// TwinCAT 3 PLC project TestIOC
// ProgramVersion: 3.1.4026.17
// libraries:
//   LCLS General, * (SLAC)
//   LCLS Vacuum, * (SLAC - LCLS)
//   lcls-twincat-common-components, * (SLAC)
//   lcls-twincat-math, * (SLAC - LCLS)
//   lcls-twincat-motion, * (SLAC)
//   lcls-twincat-optics, * (SLAC)
//   lcls-twincat-physics, * (SLAC)
//   LCLS_MotionAbstraction, * (SLAC)
//   LCLS_Tc_DevAbs, * (SLAC - LCLS)
//   PMPS, * (SLAC - LCLS)
//   Tc2_MC2, * (Beckhoff Automation GmbH)
//   Tc2_Standard, * (Beckhoff Automation GmbH)
//   Tc2_System, * (Beckhoff Automation GmbH)
//   Tc3_Module, * (Beckhoff Automation GmbH)
//   TcUnit, * (www.tcunit.org)
// project tree:
//   DUTs/ ENUM_Test.TcDUT (not stored), ST_NestedTypes01.TcDUT, ST_NestedTypes02.TcDUT, ST_NestedTypes03.TcDUT, ST_NestedTypes04.TcDUT, ST_NestedTypes05.TcDUT, ST_PytmcTypes.TcDUT (not stored)
//   GVLs/ GVL.TcGVL
//   / PlcTask.TcTTO
//   POUs/ Main.TcPOU (not stored), F_UpdateArray.TcPOU (not stored)
// real-time tasks:
//   TASK PlcTask: cycle T#10ms, priority 20, ADS port 350
// motion (NC):
//   TASK NC-Task 1 SAF: cycle T#2ms, priority 4, ADS port 501
//   TASK NC-Task 1 SVB: cycle T#10ms, priority 8, ADS port 511
//   AXIS Axis 1 (id 1)
//     OtherSettings: AllowMotionCmdToSlave=true
//     encoder EncType=1
//     drive DrvType=5
//       Analog: TorqueSetpointScale=10, ScaleFactorActTorque=0.1
//       TimeComp: TaskDelayCycles=1
//     controller CtrType=1
//       CtrPara: PriorControlFactor=1
//         Observer: BandWidth=20
//   AXIS Axis 2 (id 2)
//     OtherSettings: AllowMotionCmdToSlave=true
//     encoder EncType=1
//     drive DrvType=5
//       Analog: TorqueSetpointScale=10, ScaleFactorActTorque=0.1
//       TimeComp: TaskDelayCycles=1
//     controller CtrType=1
//       CtrPara: PriorControlFactor=1
//         Observer: BandWidth=20
//   AXIS Axis 3 (id 3)
//     OtherSettings: AllowMotionCmdToSlave=true
//     encoder EncType=1
//     drive DrvType=5
//       Analog: TorqueSetpointScale=10, ScaleFactorActTorque=0.1
//       TimeComp: TaskDelayCycles=1
//     controller CtrType=1
//       CtrPara: PriorControlFactor=1
//         Observer: BandWidth=20
//   AXIS Axis 4 (id 4)
//     OtherSettings: AllowMotionCmdToSlave=true
//     encoder EncType=1
//     drive DrvType=5
//       Analog: TorqueSetpointScale=10, ScaleFactorActTorque=0.1
//       TimeComp: TaskDelayCycles=1
//     controller CtrType=1
//       CtrPara: PriorControlFactor=1
//         Observer: BandWidth=20
//   AXIS Axis 5 (id 5)
//     OtherSettings: AllowMotionCmdToSlave=true
//     encoder EncType=1
//     drive DrvType=5
//       Analog: TorqueSetpointScale=10, ScaleFactorActTorque=0.1
//       TimeComp: TaskDelayCycles=1
//     controller CtrType=1
//       CtrPara: PriorControlFactor=1
//         Observer: BandWidth=20
//   AXIS Axis 6 (id 6)
//     OtherSettings: AllowMotionCmdToSlave=true
//     encoder EncType=1
//     drive DrvType=5
//       Analog: TorqueSetpointScale=10, ScaleFactorActTorque=0.1
//       TimeComp: TaskDelayCycles=1
//     controller CtrType=1
//       CtrPara: PriorControlFactor=1
//         Observer: BandWidth=20
//   AXIS Axis 7 (id 7)
//     OtherSettings: AllowMotionCmdToSlave=true
//     encoder EncType=1
//     drive DrvType=5
//       Analog: TorqueSetpointScale=10, ScaleFactorActTorque=0.1
//       TimeComp: TaskDelayCycles=1
//     controller CtrType=1
//       CtrPara: PriorControlFactor=1
//         Observer: BandWidth=20
//   AXIS Axis 8 (id 8)
//     OtherSettings: AllowMotionCmdToSlave=true
//     encoder EncType=1
//     drive DrvType=5
//       Analog: TorqueSetpointScale=10, ScaleFactorActTorque=0.1
//       TimeComp: TaskDelayCycles=1
//     controller CtrType=1
//       CtrPara: PriorControlFactor=1
//         Observer: BandWidth=20
//   AXIS Axis 9 (id 9)
//     OtherSettings: AllowMotionCmdToSlave=true
//     encoder EncType=1
//     drive DrvType=5
//       Analog: TorqueSetpointScale=10, ScaleFactorActTorque=0.1
//       TimeComp: TaskDelayCycles=1
//     controller CtrType=1
//       CtrPara: PriorControlFactor=1
//         Observer: BandWidth=20
//   AXIS Axis 10 (id 10)
//     OtherSettings: AllowMotionCmdToSlave=true
//     encoder EncType=1
//     drive DrvType=5
//       Analog: TorqueSetpointScale=10, ScaleFactorActTorque=0.1
//       TimeComp: TaskDelayCycles=1
//     controller CtrType=1
//       CtrPara: PriorControlFactor=1
//         Observer: BandWidth=20
//   AXIS Axis 11 (id 11)
//     OtherSettings: AllowMotionCmdToSlave=true
//     encoder EncType=1
//     drive DrvType=5
//       Analog: TorqueSetpointScale=10, ScaleFactorActTorque=0.1
//       TimeComp: TaskDelayCycles=1
//     controller CtrType=1
//       CtrPara: PriorControlFactor=1
//         Observer: BandWidth=20
//   AXIS Axis 12 (id 12)
//     OtherSettings: AllowMotionCmdToSlave=true
//     encoder EncType=1
//     drive DrvType=5
//       Analog: TorqueSetpointScale=10, ScaleFactorActTorque=0.1
//       TimeComp: TaskDelayCycles=1
//     controller CtrType=1
//       CtrPara: PriorControlFactor=1
//         Observer: BandWidth=20
//   AXIS Axis 13 (id 13)
//     OtherSettings: AllowMotionCmdToSlave=true
//     encoder EncType=1
//     drive DrvType=5
//       Analog: TorqueSetpointScale=10, ScaleFactorActTorque=0.1
//       TimeComp: TaskDelayCycles=1
//     controller CtrType=1
//       CtrPara: PriorControlFactor=1
//         Observer: BandWidth=20
//   AXIS Axis 14 (id 14)
//     OtherSettings: AllowMotionCmdToSlave=true
//     encoder EncType=1
//     drive DrvType=5
//       Analog: TorqueSetpointScale=10, ScaleFactorActTorque=0.1
//       TimeComp: TaskDelayCycles=1
//     controller CtrType=1
//       CtrPara: PriorControlFactor=1
//         Observer: BandWidth=20
//   AXIS Axis 15 (id 15)
//     OtherSettings: AllowMotionCmdToSlave=true
//     encoder EncType=1
//     drive DrvType=5
//       Analog: TorqueSetpointScale=10, ScaleFactorActTorque=0.1
//       TimeComp: TaskDelayCycles=1
//     controller CtrType=1
//       CtrPara: PriorControlFactor=1
//         Observer: BandWidth=20
//   AXIS Axis 16 (id 16)
//     OtherSettings: AllowMotionCmdToSlave=true
//     encoder EncType=1
//     drive DrvType=5
//       Analog: TorqueSetpointScale=10, ScaleFactorActTorque=0.1
//       TimeComp: TaskDelayCycles=1
//     controller CtrType=1
//       CtrPara: PriorControlFactor=1
//         Observer: BandWidth=20
//   AXIS Axis 17 (id 17)
//     OtherSettings: AllowMotionCmdToSlave=true
//     encoder EncType=1
//     drive DrvType=5
//       Analog: TorqueSetpointScale=10, ScaleFactorActTorque=0.1
//       TimeComp: TaskDelayCycles=1
//     controller CtrType=1
//       CtrPara: PriorControlFactor=1
//         Observer: BandWidth=20
//   AXIS Axis 18 (id 18)
//     OtherSettings: AllowMotionCmdToSlave=true
//     encoder EncType=1
//     drive DrvType=5
//       Analog: TorqueSetpointScale=10, ScaleFactorActTorque=0.1
//       TimeComp: TaskDelayCycles=1
//     controller CtrType=1
//       CtrPara: PriorControlFactor=1
//         Observer: BandWidth=20
//   AXIS Axis 19 (id 19)
//     OtherSettings: AllowMotionCmdToSlave=true
//     encoder EncType=1
//     drive DrvType=5
//       Analog: TorqueSetpointScale=10, ScaleFactorActTorque=0.1
//       TimeComp: TaskDelayCycles=1
//     controller CtrType=1
//       CtrPara: PriorControlFactor=1
//         Observer: BandWidth=20
//   AXIS Axis 20 (id 20)
//     OtherSettings: AllowMotionCmdToSlave=true
//     encoder EncType=1
//     drive DrvType=5
//       Analog: TorqueSetpointScale=10, ScaleFactorActTorque=0.1
//       TimeComp: TaskDelayCycles=1
//     controller CtrType=1
//       CtrPara: PriorControlFactor=1
//         Observer: BandWidth=20
//   AXIS Axis 21 (id 21)
//     OtherSettings: AllowMotionCmdToSlave=true
//     encoder EncType=1
//     drive DrvType=5
//       Analog: TorqueSetpointScale=10, ScaleFactorActTorque=0.1
//       TimeComp: TaskDelayCycles=1
//     controller CtrType=1
//       CtrPara: PriorControlFactor=1
//         Observer: BandWidth=20
//   AXIS Axis 22 (id 22)
//     OtherSettings: AllowMotionCmdToSlave=true
//     encoder EncType=1
//     drive DrvType=5
//       Analog: TorqueSetpointScale=10, ScaleFactorActTorque=0.1
//       TimeComp: TaskDelayCycles=1
//     controller CtrType=1
//       CtrPara: PriorControlFactor=1
//         Observer: BandWidth=20
//   AXIS Axis 23 (id 23)
//     OtherSettings: AllowMotionCmdToSlave=true
//     encoder EncType=1
//     drive DrvType=5
//       Analog: TorqueSetpointScale=10, ScaleFactorActTorque=0.1
//       TimeComp: TaskDelayCycles=1
//     controller CtrType=1
//       CtrPara: PriorControlFactor=1
//         Observer: BandWidth=20
//   AXIS Axis 24 (id 24)
//     OtherSettings: AllowMotionCmdToSlave=true
//     encoder EncType=1
//     drive DrvType=5
//       Analog: TorqueSetpointScale=10, ScaleFactorActTorque=0.1
//       TimeComp: TaskDelayCycles=1
//     controller CtrType=1
//       CtrPara: PriorControlFactor=1
//         Observer: BandWidth=20
//   AXIS Axis 25 (id 25)
//     OtherSettings: AllowMotionCmdToSlave=true
//     encoder EncType=1
//     drive DrvType=5
//       Analog: TorqueSetpointScale=10, ScaleFactorActTorque=0.1
//       TimeComp: TaskDelayCycles=1
//     controller CtrType=1
//       CtrPara: PriorControlFactor=1
//         Observer: BandWidth=20
//   AXIS Axis 26 (id 26)
//     OtherSettings: AllowMotionCmdToSlave=true
//     encoder EncType=1
//     drive DrvType=5
//       Analog: TorqueSetpointScale=10, ScaleFactorActTorque=0.1
//       TimeComp: TaskDelayCycles=1
//     controller CtrType=1
//       CtrPara: PriorControlFactor=1
//         Observer: BandWidth=20
//   AXIS Axis 27 (id 27)
//     OtherSettings: AllowMotionCmdToSlave=true
//     encoder EncType=1
//     drive DrvType=5
//       Analog: TorqueSetpointScale=10, ScaleFactorActTorque=0.1
//       TimeComp: TaskDelayCycles=1
//     controller CtrType=1
//       CtrPara: PriorControlFactor=1
//         Observer: BandWidth=20
//   AXIS Axis 28 (id 28)
//     OtherSettings: AllowMotionCmdToSlave=true
//     encoder EncType=1
//     drive DrvType=5
//       Analog: TorqueSetpointScale=10, ScaleFactorActTorque=0.1
//       TimeComp: TaskDelayCycles=1
//     controller CtrType=1
//       CtrPara: PriorControlFactor=1
//         Observer: BandWidth=20
//   AXIS Axis 29 (id 29)
//     OtherSettings: AllowMotionCmdToSlave=true
//     encoder EncType=1
//     drive DrvType=5
//       Analog: TorqueSetpointScale=10, ScaleFactorActTorque=0.1
//       TimeComp: TaskDelayCycles=1
//     controller CtrType=1
//       CtrPara: PriorControlFactor=1
//         Observer: BandWidth=20
//   AXIS Axis 30 (id 30)
//     OtherSettings: AllowMotionCmdToSlave=true
//     encoder EncType=1
//     drive DrvType=5
//       Analog: TorqueSetpointScale=10, ScaleFactorActTorque=0.1
//       TimeComp: TaskDelayCycles=1
//     controller CtrType=1
//       CtrPara: PriorControlFactor=1
//         Observer: BandWidth=20
//   AXIS Axis 31 (id 31)
//     OtherSettings: AllowMotionCmdToSlave=true
//     encoder EncType=1
//     drive DrvType=5
//       Analog: TorqueSetpointScale=10, ScaleFactorActTorque=0.1
//       TimeComp: TaskDelayCycles=1
//     controller CtrType=1
//       CtrPara: PriorControlFactor=1
//         Observer: BandWidth=20
//   AXIS Axis 32 (id 32)
//     OtherSettings: AllowMotionCmdToSlave=true
//     encoder EncType=1
//     drive DrvType=5
//       Analog: TorqueSetpointScale=10, ScaleFactorActTorque=0.1
//       TimeComp: TaskDelayCycles=1
//     controller CtrType=1
//       CtrPara: PriorControlFactor=1
//         Observer: BandWidth=20
//   AXIS Axis 33 (id 33)
//     OtherSettings: AllowMotionCmdToSlave=true
//     encoder EncType=1
//     drive DrvType=5
//       Analog: TorqueSetpointScale=10, ScaleFactorActTorque=0.1
//       TimeComp: TaskDelayCycles=1
//     controller CtrType=1
//       CtrPara: PriorControlFactor=1
//         Observer: BandWidth=20
//   AXIS Axis 34 (id 34)
//     OtherSettings: AllowMotionCmdToSlave=true
//     encoder EncType=1
//     drive DrvType=5
//       Analog: TorqueSetpointScale=10, ScaleFactorActTorque=0.1
//       TimeComp: TaskDelayCycles=1
//     controller CtrType=1
//       CtrPara: PriorControlFactor=1
//         Observer: BandWidth=20
//   AXIS Axis 35 (id 35)
//     OtherSettings: AllowMotionCmdToSlave=true
//     encoder EncType=1
//     drive DrvType=5
//       Analog: TorqueSetpointScale=10, ScaleFactorActTorque=0.1
//       TimeComp: TaskDelayCycles=1
//     controller CtrType=1
//       CtrPara: PriorControlFactor=1
//         Observer: BandWidth=20
//   AXIS Axis 36 (id 36)
//     OtherSettings: AllowMotionCmdToSlave=true
//     encoder EncType=1
//     drive DrvType=5
//       Analog: TorqueSetpointScale=10, ScaleFactorActTorque=0.1
//       TimeComp: TaskDelayCycles=1
//     controller CtrType=1
//       CtrPara: PriorControlFactor=1
//         Observer: BandWidth=20
//   AXIS Axis 37 (id 37)
//     OtherSettings: AllowMotionCmdToSlave=true
//     encoder EncType=1
//     drive DrvType=5
//       Analog: TorqueSetpointScale=10, ScaleFactorActTorque=0.1
//       TimeComp: TaskDelayCycles=1
//     controller CtrType=1
//       CtrPara: PriorControlFactor=1
//         Observer: BandWidth=20
//   AXIS Axis 38 (id 38)
//     OtherSettings: AllowMotionCmdToSlave=true
//     encoder EncType=1
//     drive DrvType=5
//       Analog: TorqueSetpointScale=10, ScaleFactorActTorque=0.1
//       TimeComp: TaskDelayCycles=1
//     controller CtrType=1
//       CtrPara: PriorControlFactor=1
//         Observer: BandWidth=20
//   AXIS Axis 39 (id 39)
//     OtherSettings: AllowMotionCmdToSlave=true
//     encoder EncType=1
//     drive DrvType=5
//       Analog: TorqueSetpointScale=10, ScaleFactorActTorque=0.1
//       TimeComp: TaskDelayCycles=1
//     controller CtrType=1
//       CtrPara: PriorControlFactor=1
//         Observer: BandWidth=20
//   AXIS Axis 40 (id 40)
//     OtherSettings: AllowMotionCmdToSlave=true
//     encoder EncType=1
//     drive DrvType=5
//       Analog: TorqueSetpointScale=10, ScaleFactorActTorque=0.1
//       TimeComp: TaskDelayCycles=1
//     controller CtrType=1
//       CtrPara: PriorControlFactor=1
//         Observer: BandWidth=20
//   AXIS Axis 41 (id 41)
//     OtherSettings: AllowMotionCmdToSlave=true
//     encoder EncType=1
//     drive DrvType=5
//       Analog: TorqueSetpointScale=10, ScaleFactorActTorque=0.1
//       TimeComp: TaskDelayCycles=1
//     controller CtrType=1
//       CtrPara: PriorControlFactor=1
//         Observer: BandWidth=20
//   AXIS Axis 42 (id 42)
//     OtherSettings: AllowMotionCmdToSlave=true
//     encoder EncType=1
//     drive DrvType=5
//       Analog: TorqueSetpointScale=10, ScaleFactorActTorque=0.1
//       TimeComp: TaskDelayCycles=1
//     controller CtrType=1
//       CtrPara: PriorControlFactor=1
//         Observer: BandWidth=20
//   AXIS Axis 43 (id 43)
//     OtherSettings: AllowMotionCmdToSlave=true
//     encoder EncType=1
//     drive DrvType=5
//       Analog: TorqueSetpointScale=10, ScaleFactorActTorque=0.1
//       TimeComp: TaskDelayCycles=1
//     controller CtrType=1
//       CtrPara: PriorControlFactor=1
//         Observer: BandWidth=20
//   AXIS Axis 44 (id 44)
//     OtherSettings: AllowMotionCmdToSlave=true
//     encoder EncType=1
//     drive DrvType=5
//       Analog: TorqueSetpointScale=10, ScaleFactorActTorque=0.1
//       TimeComp: TaskDelayCycles=1
//     controller CtrType=1
//       CtrPara: PriorControlFactor=1
//         Observer: BandWidth=20
//   AXIS Axis 45 (id 45)
//     OtherSettings: AllowMotionCmdToSlave=true
//     encoder EncType=1
//     drive DrvType=5
//       Analog: TorqueSetpointScale=10, ScaleFactorActTorque=0.1
//       TimeComp: TaskDelayCycles=1
//     controller CtrType=1
//       CtrPara: PriorControlFactor=1
//         Observer: BandWidth=20
//   AXIS Axis 46 (id 46)
//     OtherSettings: AllowMotionCmdToSlave=true
//     encoder EncType=1
//     drive DrvType=5
//       Analog: TorqueSetpointScale=10, ScaleFactorActTorque=0.1
//       TimeComp: TaskDelayCycles=1
//     controller CtrType=1
//       CtrPara: PriorControlFactor=1
//         Observer: BandWidth=20
//   AXIS Axis 47 (id 47)
//     OtherSettings: AllowMotionCmdToSlave=true
//     encoder EncType=1
//     drive DrvType=5
//       Analog: TorqueSetpointScale=10, ScaleFactorActTorque=0.1
//       TimeComp: TaskDelayCycles=1
//     controller CtrType=1
//       CtrPara: PriorControlFactor=1
//         Observer: BandWidth=20
//   AXIS Axis 48 (id 48)
//     OtherSettings: AllowMotionCmdToSlave=true
//     encoder EncType=1
//     drive DrvType=5
//       Analog: TorqueSetpointScale=10, ScaleFactorActTorque=0.1
//       TimeComp: TaskDelayCycles=1
//     controller CtrType=1
//       CtrPara: PriorControlFactor=1
//         Observer: BandWidth=20
//   AXIS Axis 49 (id 49)
//     OtherSettings: AllowMotionCmdToSlave=true
//     encoder EncType=1
//     drive DrvType=5
//       Analog: TorqueSetpointScale=10, ScaleFactorActTorque=0.1
//       TimeComp: TaskDelayCycles=1
//     controller CtrType=1
//       CtrPara: PriorControlFactor=1
//         Observer: BandWidth=20
//   AXIS Axis 50 (id 50)
//     OtherSettings: AllowMotionCmdToSlave=true
//     encoder EncType=1
//     drive DrvType=5
//       Analog: TorqueSetpointScale=10, ScaleFactorActTorque=0.1
//       TimeComp: TaskDelayCycles=1
//     controller CtrType=1
//       CtrPara: PriorControlFactor=1
//         Observer: BandWidth=20
//   AXIS Axis 51 (id 51)
//     OtherSettings: AllowMotionCmdToSlave=true
//     encoder EncType=1
//     drive DrvType=5
//       Analog: TorqueSetpointScale=10, ScaleFactorActTorque=0.1
//       TimeComp: TaskDelayCycles=1
//     controller CtrType=1
//       CtrPara: PriorControlFactor=1
//         Observer: BandWidth=20
//   AXIS Axis 52 (id 52)
//     OtherSettings: AllowMotionCmdToSlave=true
//     encoder EncType=1
//     drive DrvType=5
//       Analog: TorqueSetpointScale=10, ScaleFactorActTorque=0.1
//       TimeComp: TaskDelayCycles=1
//     controller CtrType=1
//       CtrPara: PriorControlFactor=1
//         Observer: BandWidth=20
// variable links:
//   (this object) <-> NC-Task 1 SAF/Axes/Axis 1
//     PlcTask Inputs/Main.M1.Axis.NcToPlc <-> Outputs/ToPlc
//     PlcTask Outputs/Main.M1.Axis.PlcToNc <-> Inputs/FromPlc
//   (this object) <-> NC-Task 1 SAF/Axes/Axis 10
//     PlcTask Inputs/Main.aAxisRef[8].NcToPlc <-> Outputs/ToPlc
//     PlcTask Outputs/Main.aAxisRef[8].PlcToNc <-> Inputs/FromPlc
//   (this object) <-> NC-Task 1 SAF/Axes/Axis 11
//     PlcTask Inputs/Main.aAxisRef[9].NcToPlc <-> Outputs/ToPlc
//     PlcTask Outputs/Main.aAxisRef[9].PlcToNc <-> Inputs/FromPlc
//   (this object) <-> NC-Task 1 SAF/Axes/Axis 12
//     PlcTask Inputs/Main.aAxisRef[10].NcToPlc <-> Outputs/ToPlc
//     PlcTask Outputs/Main.aAxisRef[10].PlcToNc <-> Inputs/FromPlc
//   (this object) <-> NC-Task 1 SAF/Axes/Axis 13
//     PlcTask Inputs/Main.aAxisRef[11].NcToPlc <-> Outputs/ToPlc
//     PlcTask Outputs/Main.aAxisRef[11].PlcToNc <-> Inputs/FromPlc
//   (this object) <-> NC-Task 1 SAF/Axes/Axis 14
//     PlcTask Inputs/Main.aAxisRef[12].NcToPlc <-> Outputs/ToPlc
//     PlcTask Outputs/Main.aAxisRef[12].PlcToNc <-> Inputs/FromPlc
//   (this object) <-> NC-Task 1 SAF/Axes/Axis 15
//     PlcTask Inputs/Main.aAxisRef[13].NcToPlc <-> Outputs/ToPlc
//     PlcTask Outputs/Main.aAxisRef[13].PlcToNc <-> Inputs/FromPlc
//   (this object) <-> NC-Task 1 SAF/Axes/Axis 16
//     PlcTask Inputs/Main.aAxisRef[14].NcToPlc <-> Outputs/ToPlc
//     PlcTask Outputs/Main.aAxisRef[14].PlcToNc <-> Inputs/FromPlc
//   (this object) <-> NC-Task 1 SAF/Axes/Axis 17
//     PlcTask Inputs/Main.aAxisRef[15].NcToPlc <-> Outputs/ToPlc
//     PlcTask Outputs/Main.aAxisRef[15].PlcToNc <-> Inputs/FromPlc
//   (this object) <-> NC-Task 1 SAF/Axes/Axis 18
//     PlcTask Inputs/Main.aAxisRef[16].NcToPlc <-> Outputs/ToPlc
//     PlcTask Outputs/Main.aAxisRef[16].PlcToNc <-> Inputs/FromPlc
//   (this object) <-> NC-Task 1 SAF/Axes/Axis 19
//     PlcTask Inputs/Main.aAxisRef[17].NcToPlc <-> Outputs/ToPlc
//     PlcTask Outputs/Main.aAxisRef[17].PlcToNc <-> Inputs/FromPlc
//   (this object) <-> NC-Task 1 SAF/Axes/Axis 2
//     PlcTask Inputs/Main.M2.Axis.NcToPlc <-> Outputs/ToPlc
//     PlcTask Outputs/Main.M2.Axis.PlcToNc <-> Inputs/FromPlc
//   (this object) <-> NC-Task 1 SAF/Axes/Axis 20
//     PlcTask Inputs/Main.aAxisRef[18].NcToPlc <-> Outputs/ToPlc
//     PlcTask Outputs/Main.aAxisRef[18].PlcToNc <-> Inputs/FromPlc
//   (this object) <-> NC-Task 1 SAF/Axes/Axis 21
//     PlcTask Inputs/Main.aAxisRef[19].NcToPlc <-> Outputs/ToPlc
//     PlcTask Outputs/Main.aAxisRef[19].PlcToNc <-> Inputs/FromPlc
//   (this object) <-> NC-Task 1 SAF/Axes/Axis 22
//     PlcTask Inputs/Main.aAxisRef[20].NcToPlc <-> Outputs/ToPlc
//     PlcTask Outputs/Main.aAxisRef[20].PlcToNc <-> Inputs/FromPlc
//   (this object) <-> NC-Task 1 SAF/Axes/Axis 23
//     PlcTask Inputs/Main.aAxisRef[21].NcToPlc <-> Outputs/ToPlc
//     PlcTask Outputs/Main.aAxisRef[21].PlcToNc <-> Inputs/FromPlc
//   (this object) <-> NC-Task 1 SAF/Axes/Axis 24
//     PlcTask Inputs/Main.aAxisRef[22].NcToPlc <-> Outputs/ToPlc
//     PlcTask Outputs/Main.aAxisRef[22].PlcToNc <-> Inputs/FromPlc
//   (this object) <-> NC-Task 1 SAF/Axes/Axis 25
//     PlcTask Inputs/Main.aAxisRef[23].NcToPlc <-> Outputs/ToPlc
//     PlcTask Outputs/Main.aAxisRef[23].PlcToNc <-> Inputs/FromPlc
//   (this object) <-> NC-Task 1 SAF/Axes/Axis 26
//     PlcTask Inputs/Main.aAxisRef[24].NcToPlc <-> Outputs/ToPlc
//     PlcTask Outputs/Main.aAxisRef[24].PlcToNc <-> Inputs/FromPlc
//   (this object) <-> NC-Task 1 SAF/Axes/Axis 27
//     PlcTask Inputs/Main.aAxisRef[25].NcToPlc <-> Outputs/ToPlc
//     PlcTask Outputs/Main.aAxisRef[25].PlcToNc <-> Inputs/FromPlc
//   (this object) <-> NC-Task 1 SAF/Axes/Axis 28
//     PlcTask Inputs/Main.aAxisRef[26].NcToPlc <-> Outputs/ToPlc
//     PlcTask Outputs/Main.aAxisRef[26].PlcToNc <-> Inputs/FromPlc
//   (this object) <-> NC-Task 1 SAF/Axes/Axis 29
//     PlcTask Inputs/Main.aAxisRef[27].NcToPlc <-> Outputs/ToPlc
//     PlcTask Outputs/Main.aAxisRef[27].PlcToNc <-> Inputs/FromPlc
//   (this object) <-> NC-Task 1 SAF/Axes/Axis 3
//     PlcTask Inputs/Main.aAxisRef[1].NcToPlc <-> Outputs/ToPlc
//     PlcTask Outputs/Main.aAxisRef[1].PlcToNc <-> Inputs/FromPlc
//   (this object) <-> NC-Task 1 SAF/Axes/Axis 30
//     PlcTask Inputs/Main.aAxisRef[28].NcToPlc <-> Outputs/ToPlc
//     PlcTask Outputs/Main.aAxisRef[28].PlcToNc <-> Inputs/FromPlc
//   (this object) <-> NC-Task 1 SAF/Axes/Axis 31
//     PlcTask Inputs/Main.aAxisRef[29].NcToPlc <-> Outputs/ToPlc
//     PlcTask Outputs/Main.aAxisRef[29].PlcToNc <-> Inputs/FromPlc
//   (this object) <-> NC-Task 1 SAF/Axes/Axis 32
//     PlcTask Inputs/Main.aAxisRef[30].NcToPlc <-> Outputs/ToPlc
//     PlcTask Outputs/Main.aAxisRef[30].PlcToNc <-> Inputs/FromPlc
//   (this object) <-> NC-Task 1 SAF/Axes/Axis 33
//     PlcTask Inputs/Main.aAxisRef[31].NcToPlc <-> Outputs/ToPlc
//     PlcTask Outputs/Main.aAxisRef[31].PlcToNc <-> Inputs/FromPlc
//   (this object) <-> NC-Task 1 SAF/Axes/Axis 34
//     PlcTask Inputs/Main.aAxisRef[32].NcToPlc <-> Outputs/ToPlc
//     PlcTask Outputs/Main.aAxisRef[32].PlcToNc <-> Inputs/FromPlc
//   (this object) <-> NC-Task 1 SAF/Axes/Axis 35
//     PlcTask Inputs/Main.aAxisRef[33].NcToPlc <-> Outputs/ToPlc
//     PlcTask Outputs/Main.aAxisRef[33].PlcToNc <-> Inputs/FromPlc
//   (this object) <-> NC-Task 1 SAF/Axes/Axis 36
//     PlcTask Inputs/Main.aAxisRef[34].NcToPlc <-> Outputs/ToPlc
//     PlcTask Outputs/Main.aAxisRef[34].PlcToNc <-> Inputs/FromPlc
//   (this object) <-> NC-Task 1 SAF/Axes/Axis 37
//     PlcTask Inputs/Main.aAxisRef[35].NcToPlc <-> Outputs/ToPlc
//     PlcTask Outputs/Main.aAxisRef[35].PlcToNc <-> Inputs/FromPlc
//   (this object) <-> NC-Task 1 SAF/Axes/Axis 38
//     PlcTask Inputs/Main.aAxisRef[36].NcToPlc <-> Outputs/ToPlc
//     PlcTask Outputs/Main.aAxisRef[36].PlcToNc <-> Inputs/FromPlc
//   (this object) <-> NC-Task 1 SAF/Axes/Axis 39
//     PlcTask Inputs/Main.aAxisRef[37].NcToPlc <-> Outputs/ToPlc
//     PlcTask Outputs/Main.aAxisRef[37].PlcToNc <-> Inputs/FromPlc
//   (this object) <-> NC-Task 1 SAF/Axes/Axis 4
//     PlcTask Inputs/Main.aAxisRef[2].NcToPlc <-> Outputs/ToPlc
//     PlcTask Outputs/Main.aAxisRef[2].PlcToNc <-> Inputs/FromPlc
//   (this object) <-> NC-Task 1 SAF/Axes/Axis 40
//     PlcTask Inputs/Main.aAxisRef[38].NcToPlc <-> Outputs/ToPlc
//     PlcTask Outputs/Main.aAxisRef[38].PlcToNc <-> Inputs/FromPlc
//   (this object) <-> NC-Task 1 SAF/Axes/Axis 41
//     PlcTask Inputs/Main.aAxisRef[39].NcToPlc <-> Outputs/ToPlc
//     PlcTask Outputs/Main.aAxisRef[39].PlcToNc <-> Inputs/FromPlc
//   (this object) <-> NC-Task 1 SAF/Axes/Axis 42
//     PlcTask Inputs/Main.aAxisRef[40].NcToPlc <-> Outputs/ToPlc
//     PlcTask Outputs/Main.aAxisRef[40].PlcToNc <-> Inputs/FromPlc
//   (this object) <-> NC-Task 1 SAF/Axes/Axis 43
//     PlcTask Inputs/Main.aAxisRef[41].NcToPlc <-> Outputs/ToPlc
//     PlcTask Outputs/Main.aAxisRef[41].PlcToNc <-> Inputs/FromPlc
//   (this object) <-> NC-Task 1 SAF/Axes/Axis 44
//     PlcTask Inputs/Main.aAxisRef[42].NcToPlc <-> Outputs/ToPlc
//     PlcTask Outputs/Main.aAxisRef[42].PlcToNc <-> Inputs/FromPlc
//   (this object) <-> NC-Task 1 SAF/Axes/Axis 45
//     PlcTask Inputs/Main.aAxisRef[43].NcToPlc <-> Outputs/ToPlc
//     PlcTask Outputs/Main.aAxisRef[43].PlcToNc <-> Inputs/FromPlc
//   (this object) <-> NC-Task 1 SAF/Axes/Axis 46
//     PlcTask Inputs/Main.aAxisRef[44].NcToPlc <-> Outputs/ToPlc
//     PlcTask Outputs/Main.aAxisRef[44].PlcToNc <-> Inputs/FromPlc
//   (this object) <-> NC-Task 1 SAF/Axes/Axis 47
//     PlcTask Inputs/Main.aAxisRef[45].NcToPlc <-> Outputs/ToPlc
//     PlcTask Outputs/Main.aAxisRef[45].PlcToNc <-> Inputs/FromPlc
//   (this object) <-> NC-Task 1 SAF/Axes/Axis 48
//     PlcTask Inputs/Main.aAxisRef[46].NcToPlc <-> Outputs/ToPlc
//     PlcTask Outputs/Main.aAxisRef[46].PlcToNc <-> Inputs/FromPlc
//   (this object) <-> NC-Task 1 SAF/Axes/Axis 49
//     PlcTask Inputs/Main.aAxisRef[47].NcToPlc <-> Outputs/ToPlc
//     PlcTask Outputs/Main.aAxisRef[47].PlcToNc <-> Inputs/FromPlc
//   (this object) <-> NC-Task 1 SAF/Axes/Axis 5
//     PlcTask Inputs/Main.aAxisRef[3].NcToPlc <-> Outputs/ToPlc
//     PlcTask Outputs/Main.aAxisRef[3].PlcToNc <-> Inputs/FromPlc
//   (this object) <-> NC-Task 1 SAF/Axes/Axis 50
//     PlcTask Inputs/Main.aAxisRef[48].NcToPlc <-> Outputs/ToPlc
//     PlcTask Outputs/Main.aAxisRef[48].PlcToNc <-> Inputs/FromPlc
//   (this object) <-> NC-Task 1 SAF/Axes/Axis 51
//     PlcTask Inputs/Main.aAxisRef[49].NcToPlc <-> Outputs/ToPlc
//     PlcTask Outputs/Main.aAxisRef[49].PlcToNc <-> Inputs/FromPlc
//   (this object) <-> NC-Task 1 SAF/Axes/Axis 52
//     PlcTask Inputs/Main.aAxisRef[50].NcToPlc <-> Outputs/ToPlc
//     PlcTask Outputs/Main.aAxisRef[50].PlcToNc <-> Inputs/FromPlc
//   (this object) <-> NC-Task 1 SAF/Axes/Axis 6
//     PlcTask Inputs/Main.aAxisRef[4].NcToPlc <-> Outputs/ToPlc
//     PlcTask Outputs/Main.aAxisRef[4].PlcToNc <-> Inputs/FromPlc
//   (this object) <-> NC-Task 1 SAF/Axes/Axis 7
//     PlcTask Inputs/Main.aAxisRef[5].NcToPlc <-> Outputs/ToPlc
//     PlcTask Outputs/Main.aAxisRef[5].PlcToNc <-> Inputs/FromPlc
//   (this object) <-> NC-Task 1 SAF/Axes/Axis 8
//     PlcTask Inputs/Main.aAxisRef[6].NcToPlc <-> Outputs/ToPlc
//     PlcTask Outputs/Main.aAxisRef[6].PlcToNc <-> Inputs/FromPlc
//   (this object) <-> NC-Task 1 SAF/Axes/Axis 9
//     PlcTask Inputs/Main.aAxisRef[7].NcToPlc <-> Outputs/ToPlc
//     PlcTask Outputs/Main.aAxisRef[7].PlcToNc <-> Inputs/FromPlc

CONFIGURATION TestIOC
    RESOURCE PLC ON TwinCAT3
        TASK PlcTask(INTERVAL := T#10ms, PRIORITY := 20);
        PROGRAM Main WITH PlcTask : Main;
    END_RESOURCE
END_CONFIGURATION

// ---- DUTs/ST_NestedTypes01.TcDUT

TYPE ST_NestedTypes01 :
STRUCT
	stPytmcTypes : ST_PytmcTypes;
	stNestedTypes : ST_NestedTypes02;
END_STRUCT
END_TYPE

// ---- DUTs/ST_NestedTypes02.TcDUT

TYPE ST_NestedTypes02 :
STRUCT
	stPytmcTypes : ST_PytmcTypes;
	stNestedTypes : ST_NestedTypes03;
END_STRUCT
END_TYPE

// ---- DUTs/ST_NestedTypes03.TcDUT

TYPE ST_NestedTypes03 :
STRUCT
	stPytmcTypes : ST_PytmcTypes;
	stNestedTypes : ST_NestedTypes04;
END_STRUCT
END_TYPE

// ---- DUTs/ST_NestedTypes04.TcDUT

TYPE ST_NestedTypes04 :
STRUCT
	stPytmcTypes : ST_PytmcTypes;
	stNestedTypes : ST_NestedTypes05;
END_STRUCT
END_TYPE

// ---- DUTs/ST_NestedTypes05.TcDUT

TYPE ST_NestedTypes05 :
STRUCT
	stPytmcTypes : ST_PytmcTypes;
END_STRUCT
END_TYPE

// ---- GVLs/GVL.TcGVL

{attribute 'qualified_only'}
VAR_GLOBAL CONSTANT
	nPytmcTypesArrayLength : UINT := 99;
END_VAR
